Yaskawa INFORM job: SPHERE1.JBI

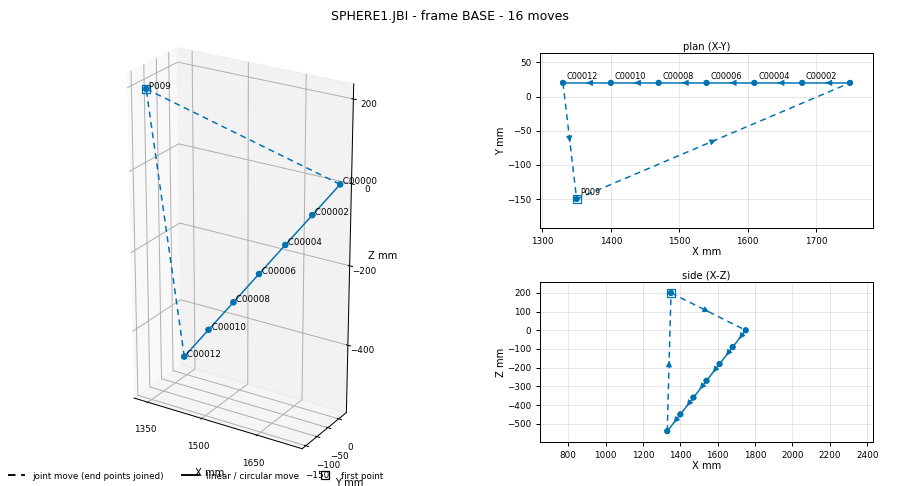
[picture p0: tool path of SPHERE1.JBI in frame BASE, 16 of 16 moves have a stored position in this frame; points joined in program order, loops and branches not executed]
/JOB
//NAME SPHERE1
//POS
///NPOS 14,0,14,1,0,1
///TOOL 0
///POSTYPE BASE
///RECTAN
///RCONF 0,0,0,0,0,0,0,0,0,0,0,0,0,0,0,0,0,0,0,0,0,0,0,0
C00000=1750.000,20.000,0.000,-178.0000,-30.0000,0.0000
C00001=1750.000,20.000,0.000,-178.0000,-30.0000,0.0000
C00002=1680.000,20.000,-90.000,-178.0000,-40.0000,0.0000
C00003=1680.000,20.000,-90.000,-178.0000,-40.0000,0.0000
C00004=1610.000,20.000,-180.000,-178.0000,-50.0000,0.0000
C00005=1610.000,20.000,-180.000,-178.0000,-50.0000,0.0000
C00006=1540.000,20.000,-270.000,-178.0000,-60.0000,0.0000
C00007=1540.000,20.000,-270.000,-178.0000,-60.0000,0.0000
C00008=1470.000,20.000,-360.000,-178.0000,-70.0000,0.0000
C00009=1470.000,20.000,-360.000,-178.0000,-70.0000,0.0000
C00010=1400.000,20.000,-450.000,-178.0000,-80.0000,0.0000
C00011=1400.000,20.000,-450.000,-178.0000,-80.0000,0.0000
C00012=1330.000,20.000,-540.000,-178.0000,-90.0000,0.0000
C00013=1330.000,20.000,-540.000,-178.0000,-90.0000,0.0000
///POSTYPE PULSE
///PULSE
EC00000=0
EC00001=368640
EC00002=368640
EC00003=0
EC00004=0
EC00005=368640
EC00006=368640
EC00007=0
EC00008=0
EC00009=368640
EC00010=368640
EC00011=0
EC00012=0
EC00013=368640
///POSTYPE BASE
///RECTAN
///RCONF 1,0,0,0,0,0,0,0,0,0,0,0,0,0,0,0,0,0,0,0,0,0,0,0
P00009=1350.000,-150.000,200.000,-180.0000,-45.0000,0.0000
///POSTYPE PULSE
///PULSE
EX00000=0
//INST
///DATE 2023/02/09 12:01
///ATTR SC,RW,RJ
////FRAME BASE
///GROUP1 RB1,ST1
NOP
MOVJ P009 EX000 VJ=15.00
MOVJ C00000 EC00000 VJ=15.00
CALL JOB:SPYON
MOVJ C00001 EC00001 VJ=10.00
MOVC C00002 EC00002 V=150.0
MOVJ C00003 EC00003 VJ=10.00
MOVC C00004 EC00004 V=150.0
MOVJ C00005 EC00005 VJ=10.00
MOVC C00006 EC00006 V=150.0
MOVJ C00007 EC00007 VJ=10.00
MOVC C00008 EC00008 V=150.0
MOVJ C00009 EC00009 VJ=10.00
MOVC C00010 EC00010 V=150.0
MOVJ C00011 EC00011 VJ=10.00
MOVC C00012 EC00012 V=150.0
MOVJ C00013 EC00013 VJ=10.00
CALL JOB:SPYOF
MOVJ P009 EX000 VJ=15.00
END
